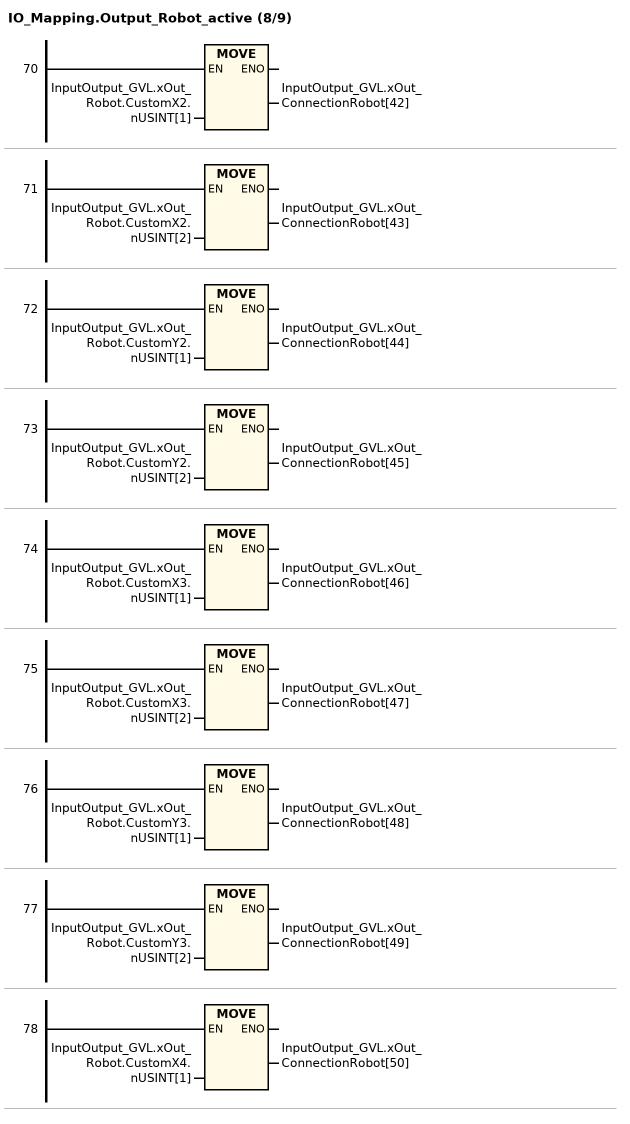
// NETWORK 70
InputOutput_GVL.xOut_ConnectionRobot[42] := InputOutput_GVL.xOut_Robot.CustomX2.nUSINT[1];

// NETWORK 71
InputOutput_GVL.xOut_ConnectionRobot[43] := InputOutput_GVL.xOut_Robot.CustomX2.nUSINT[2];

// NETWORK 72
InputOutput_GVL.xOut_ConnectionRobot[44] := InputOutput_GVL.xOut_Robot.CustomY2.nUSINT[1];

// NETWORK 73
InputOutput_GVL.xOut_ConnectionRobot[45] := InputOutput_GVL.xOut_Robot.CustomY2.nUSINT[2];

// NETWORK 74
InputOutput_GVL.xOut_ConnectionRobot[46] := InputOutput_GVL.xOut_Robot.CustomX3.nUSINT[1];

// NETWORK 75
InputOutput_GVL.xOut_ConnectionRobot[47] := InputOutput_GVL.xOut_Robot.CustomX3.nUSINT[2];

// NETWORK 76
InputOutput_GVL.xOut_ConnectionRobot[48] := InputOutput_GVL.xOut_Robot.CustomY3.nUSINT[1];

// NETWORK 77
InputOutput_GVL.xOut_ConnectionRobot[49] := InputOutput_GVL.xOut_Robot.CustomY3.nUSINT[2];

// NETWORK 78
InputOutput_GVL.xOut_ConnectionRobot[50] := InputOutput_GVL.xOut_Robot.CustomX4.nUSINT[1];

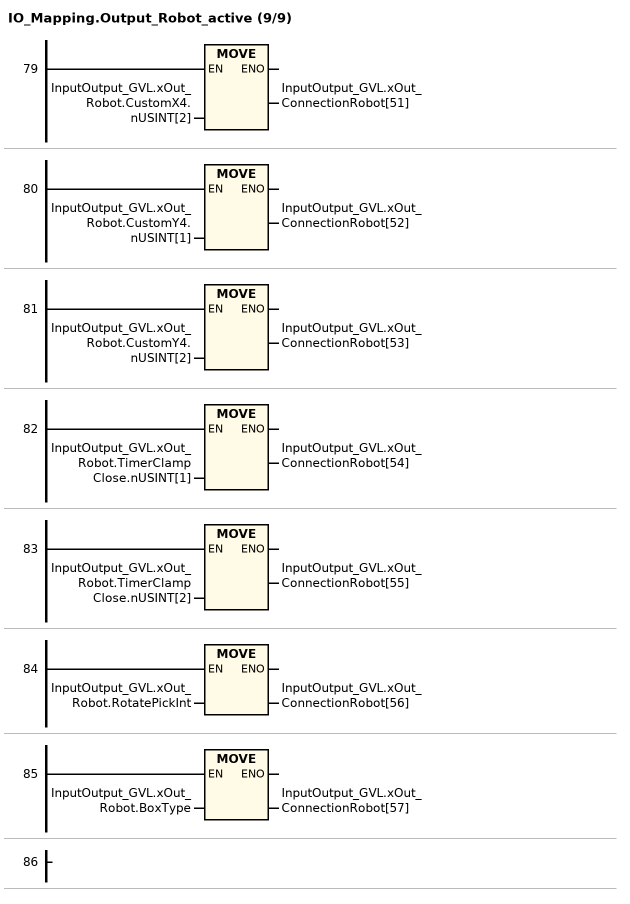
// NETWORK 79
InputOutput_GVL.xOut_ConnectionRobot[51] := InputOutput_GVL.xOut_Robot.CustomX4.nUSINT[2];

// NETWORK 80
InputOutput_GVL.xOut_ConnectionRobot[52] := InputOutput_GVL.xOut_Robot.CustomY4.nUSINT[1];

// NETWORK 81
InputOutput_GVL.xOut_ConnectionRobot[53] := InputOutput_GVL.xOut_Robot.CustomY4.nUSINT[2];

// NETWORK 82
InputOutput_GVL.xOut_ConnectionRobot[54] := InputOutput_GVL.xOut_Robot.TimerClampClose.nUSINT[1];

// NETWORK 83
InputOutput_GVL.xOut_ConnectionRobot[55] := InputOutput_GVL.xOut_Robot.TimerClampClose.nUSINT[2];

// NETWORK 84
InputOutput_GVL.xOut_ConnectionRobot[56] := InputOutput_GVL.xOut_Robot.RotatePickInt;

// NETWORK 85
InputOutput_GVL.xOut_ConnectionRobot[57] := InputOutput_GVL.xOut_Robot.BoxType;

// NETWORK 86
END_ACTION

END_PROGRAM

(* stored: Version 1.1.0.1, ProductVersion 3.1.4024.12
   POU IO_Mapping: Id {d4dc24a6-4159-49d8-be23-5d63393257fa}, SpecialFunc None
   Action Input_Button_active: Id {70efb88d-f7ec-436f-b340-952041209401}
   Action Input_Feedback_active: Id {43634fe0-7808-457a-935d-c3df193253d2}
   Action Input_Interlock_active: Id {1642d3d1-314a-4671-b469-12623cd0d8bb}
   Action Input_LimitSwitch_active: Id {34ef6b74-438e-496d-bede-0bee70b5d751}
   Action Input_Proximity_active: Id {f852badd-7863-4e11-8c61-01ef336cad9d}
   Action Input_Reedswitch_active: Id {eec07759-d078-4434-be6a-49e3c8f42fae}
   Action Input_Robot_active: Id {ca23446f-245a-439c-a341-fe7a53fd875b}
   Action Input_Safety_active: Id {43d33566-8903-467c-991e-b9da4252c007}
   Action Input_Sensor_active: Id {c6393cc3-b05e-45a5-a291-ec9453a4c311}
   Action Output_Indicator_active: Id {b1592667-1850-477f-b88d-ed14c49c91ca}
   Action Output_Interlock_active: Id {e662cbdc-9a3c-4454-b716-13fe633ba940}
   Action Output_Motor_active: Id {9ba163c9-fc33-42f4-b269-c3ca5b5c4a31}
   Action Output_Pneumatic_active: Id {bbe5ee44-6b9d-484d-a98a-559fe40e55e4}
   Action Output_Robot_active: Id {41c70136-13fc-40e1-892d-f8d5c142a919} *)
